{attribute 'Tc2GvlVarNames'}
VAR_GLOBAL CONSTANT
	(* KKKW_Zustand_Status *)
	E_KKKW_Zustand_Status_Idle_Sperre				: SINT := 0;
	E_KKKW_Zustand_Status_Betriebsbereit			: SINT := 1;
	E_KKKW_Zustand_Status_Nachl						: SINT := 2;
	E_KKKW_Zustand_Status_Vorl						: SINT := 3;
	E_KKKW_Zustand_Status_Betrieb					: SINT := 4;
	E_KKKW_Zustand_Status_Betrieb_Sperre			: SINT := 5;
	E_KKKW_Zustand_Status_Stoerung					: SINT := 99;

	(* System_KKKW_Zustand_Status *)
	E_System_KKKW_Zustand_Status_Idle_Sperre		: SINT := 0;
	E_System_KKKW_Zustand_Status_Betriebsbereit		: SINT := 1;
	E_System_KKKW_Zustand_Status_Nachl_Stellventil	: SINT := 2;
	E_System_KKKW_Zustand_Status_Vorl_Stellventil	: SINT := 3;
	E_System_KKKW_Zustand_Status_Nachl_Pumpe		: SINT := 4;
	E_System_KKKW_Zustand_Status_Vorl_Pumpe			: SINT := 5;
	(*E_System_KKKW_Zustand_Status_Nachl_KKKW		: SINT := 6;
	E_System_KKKW_Zustand_Status_Vorl_KKKW			: SINT := 7;	*)
	E_System_KKKW_Zustand_Status_Betrieb			: SINT := 8;
	E_System_KKKW_Zustand_Status_Betrieb_Sperre		: SINT := 9;
	E_System_KKKW_Zustand_Status_Stoerung			: SINT := 99;
END_VAR

(* stored: Version 1.1.0.1, ProductVersion 3.1.4024.9
   GVL Con_KKKW: Id {111eef6b-c0bc-4d54-91c3-ce6685bb8eec} *)
